Yaskawa INFORM job: PAUSE.JBI

/JOB
//NAME PAUSE
//POS
///NPOS 3,0,0,0,0,0
///TOOL 0
///POSTYPE PULSE
///PULSE
C00000=-63951,-155157,126850,-105314,-81596,-126669
C00001=-98085,-155157,126850,-105314,-81596,-126669
C00002=-63951,-155157,126850,-105314,-81596,-126669
//INST
///DATE 2022/03/01 09:37
///ATTR SC,RW
///GROUP1 RB1
NOP
CALL JOB:SYS_VERIFY_GATE_LOCKED
MOVJ C00000 VJ=65.00  //HOME
MOVJ C00001 VJ=65.00
CALL JOB:SYS_UNLOCK_GATE
PAUSE
MOVJ C00002 VJ=65.00  //HOME
END
